# EPICS substitutions: sr570/iocBoot/iocsr570/sr570.substitutions
file "SR570.db"
{
pattern
{P,             A,  PORT}
{"BL:SR570_1:", "", "SR570_1"}
{"BL:SR570_2:", "", "SR570_2"}
{"BL:SR570_3:", "", "SR570_3"}
{"BL:SR570_4:", "", "SR570_4"}
{"BL:SR570_5:", "", "SR570_5"}
{"BL:SR570_6:", "", "SR570_6"}
{"BL:SR570_7:", "", "SR570_7"}
{"BL:SR570_8:", "", "SR570_8"}
}
